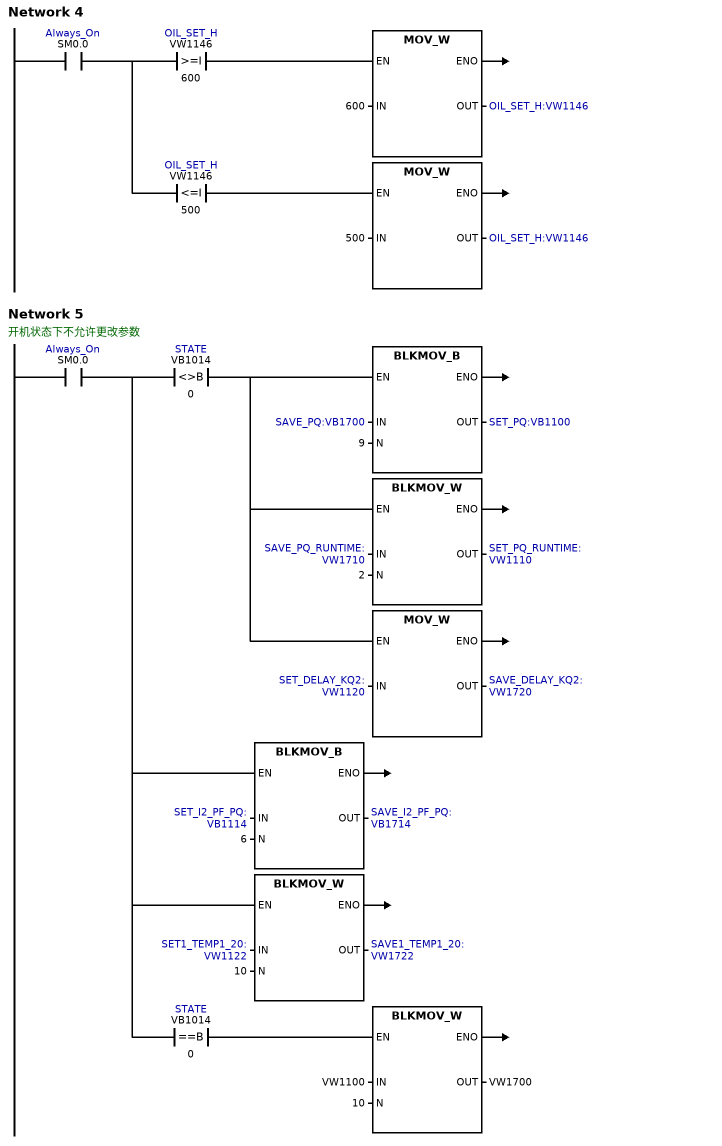
[picture p48: SBR5 networks 4-5]
Network 4
LD     Always_On:SM0.0
LPS
AW>=   OIL_SET_H:VW1146, 600
MOVW   600, OIL_SET_H:VW1146
LPP
AW<=   OIL_SET_H:VW1146, 500
MOVW   500, OIL_SET_H:VW1146
Network 5
// 开机状态下不允许更改参数
LD     Always_On:SM0.0
LPS
AB<>   STATE:VB1014, 0
BMB    SAVE_PQ:VB1700, SET_PQ:VB1100, 9
BMW    SAVE_PQ_RUNTIME:VW1710, SET_PQ_RUNTIME:VW1110, 2
MOVW   SET_DELAY_KQ2:VW1120, SAVE_DELAY_KQ2:VW1720
LPP
BMB    SET_I2_PF_PQ:VB1114, SAVE_I2_PF_PQ:VB1714, 6
BMW    SET1_TEMP1_20:VW1122, SAVE1_TEMP1_20:VW1722, 10
AB=    STATE:VB1014, 0
BMW    VW1100, VW1700, 10
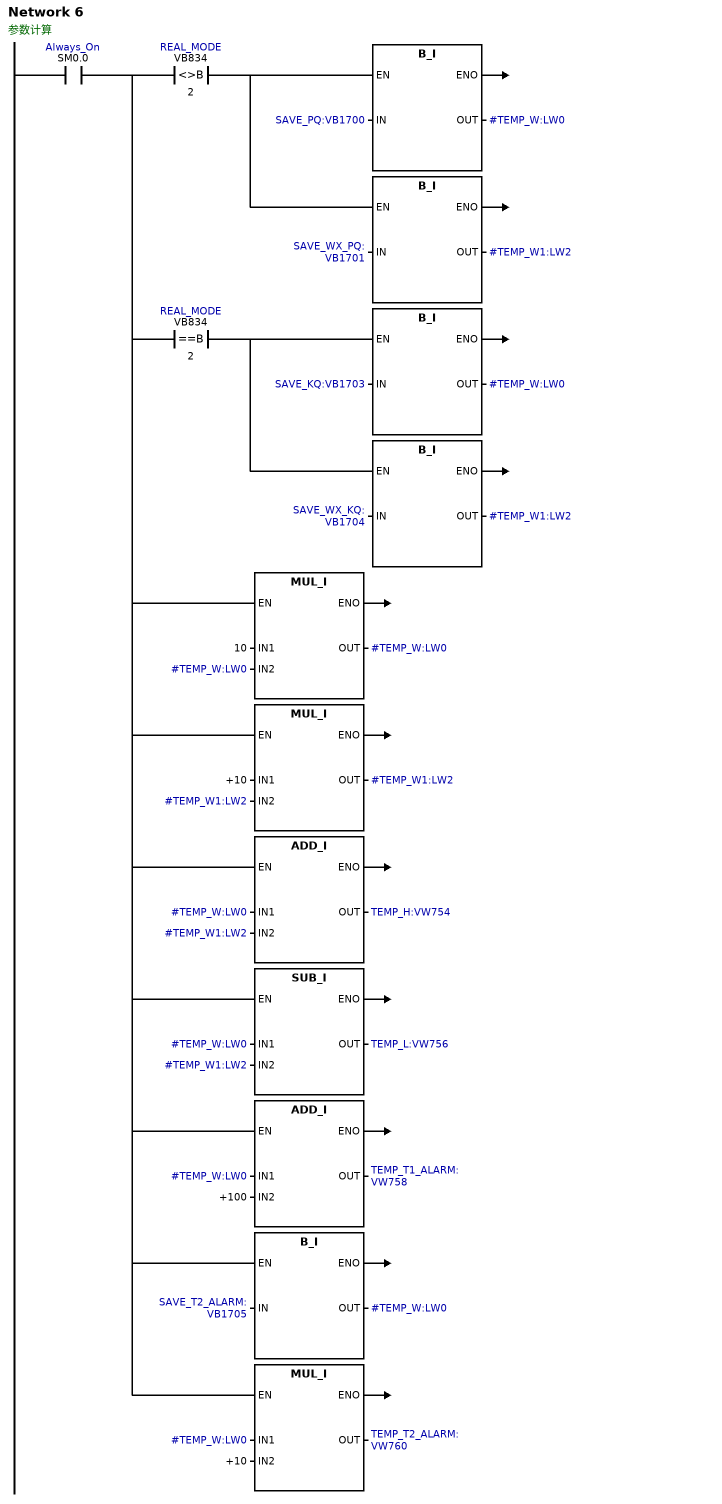
Network 6
// 参数计算
LD     Always_On:SM0.0
LPS
AB<>   REAL_MODE:VB834, 2
BTI    SAVE_PQ:VB1700, #TEMP_W:LW0
BTI    SAVE_WX_PQ:VB1701, #TEMP_W1:LW2
LRD
AB=    REAL_MODE:VB834, 2
BTI    SAVE_KQ:VB1703, #TEMP_W:LW0
BTI    SAVE_WX_KQ:VB1704, #TEMP_W1:LW2
LPP
*I     10, #TEMP_W:LW0
*I     +10, #TEMP_W1:LW2
MOVW   #TEMP_W:LW0, TEMP_H:VW754
+I     #TEMP_W1:LW2, TEMP_H:VW754
MOVW   #TEMP_W:LW0, TEMP_L:VW756
-I     #TEMP_W1:LW2, TEMP_L:VW756
MOVW   #TEMP_W:LW0, TEMP_T1_ALARM:VW758
+I     +100, TEMP_T1_ALARM:VW758
BTI    SAVE_T2_ALARM:VB1705, #TEMP_W:LW0
MOVW   #TEMP_W:LW0, TEMP_T2_ALARM:VW760
*I     +10, TEMP_T2_ALARM:VW760
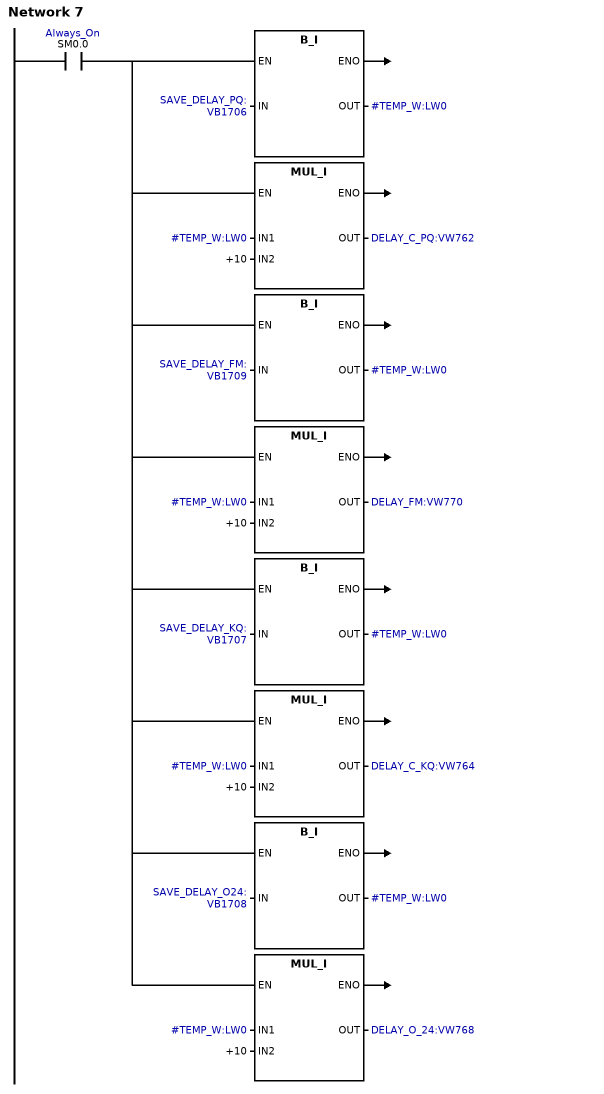
Network 7
LD     Always_On:SM0.0
BTI    SAVE_DELAY_PQ:VB1706, #TEMP_W:LW0
MOVW   #TEMP_W:LW0, DELAY_C_PQ:VW762
*I     +10, DELAY_C_PQ:VW762
BTI    SAVE_DELAY_FM:VB1709, #TEMP_W:LW0
MOVW   #TEMP_W:LW0, DELAY_FM:VW770
*I     +10, DELAY_FM:VW770
BTI    SAVE_DELAY_KQ:VB1707, #TEMP_W:LW0
MOVW   #TEMP_W:LW0, DELAY_C_KQ:VW764
*I     +10, DELAY_C_KQ:VW764
BTI    SAVE_DELAY_O24:VB1708, #TEMP_W:LW0
MOVW   #TEMP_W:LW0, DELAY_O_24:VW768
*I     +10, DELAY_O_24:VW768
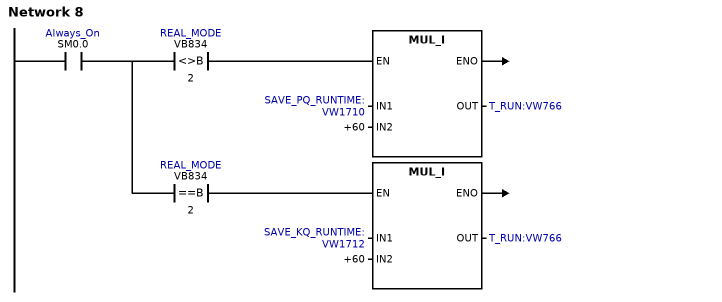
Network 8
LD     Always_On:SM0.0
LPS
AB<>   REAL_MODE:VB834, 2
MOVW   SAVE_PQ_RUNTIME:VW1710, T_RUN:VW766
*I     +60, T_RUN:VW766
LPP
AB=    REAL_MODE:VB834, 2
MOVW   SAVE_KQ_RUNTIME:VW1712, T_RUN:VW766
*I     +60, T_RUN:VW766
END_SUBROUTINE_BLOCK

SUBROUTINE_BLOCK 温度采样:SBR6
TITLE=
VAR_INPUT
ADDRESS:DWORD;	// LD0 
IN:WORD;	// LW4 
IN_TEMP:WORD;	// LW6 
F_SET:BOOL;	// L8.0 
END_VAR
VAR_OUTPUT
OUT:WORD;	// LW9 
AVERAGE:WORD;	// LW11 
OUT_TEMP:WORD;	// LW13 
END_VAR
VAR
MAX:WORD;	// LW15 
MIN:WORD;	// LW17 
TEMP_B:BYTE;	// LB19 
TEMP_W:WORD;	// LW20 
TEMP_DW:DWORD;	// LD22 
SUM:DWORD;	// LD26 
PP1:DWORD;	// LD30 
PP2:DWORD;	// LD34 
TEMP_W2:WORD;	// LW38 
AC_TEMP:DWORD;	// LD40 
END_VAR
BEGIN
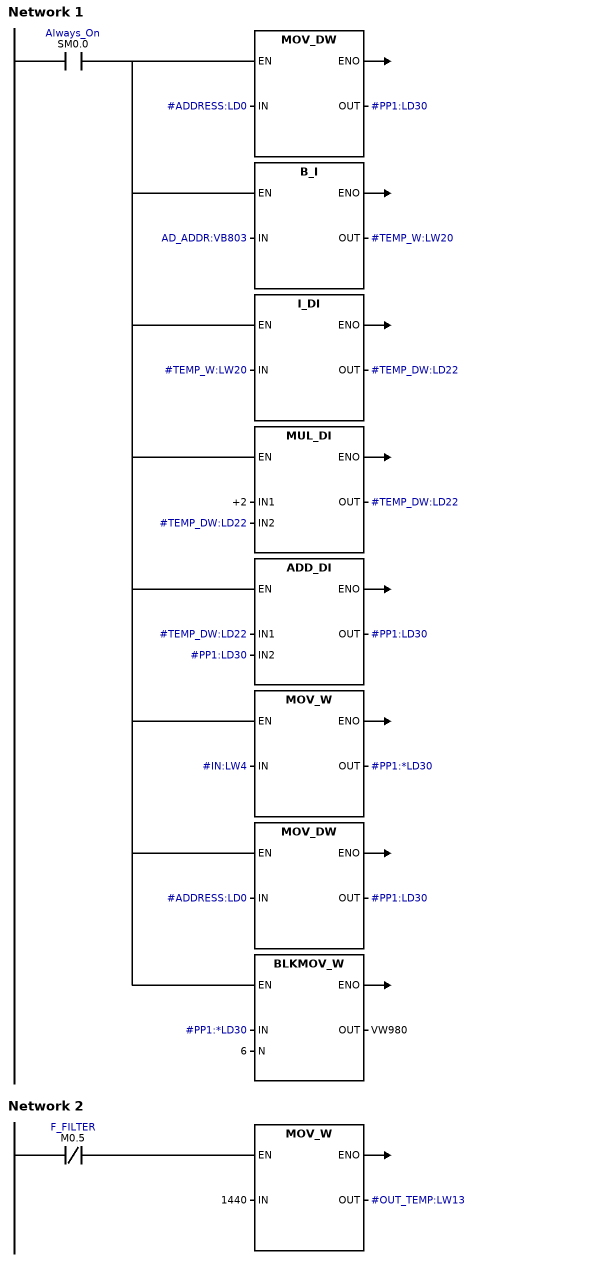
Network 1
LD     Always_On:SM0.0
MOVD   #ADDRESS:LD0, #PP1:LD30
BTI    AD_ADDR:VB803, #TEMP_W:LW20
ITD    #TEMP_W:LW20, #TEMP_DW:LD22
*D     +2, #TEMP_DW:LD22
+D     #TEMP_DW:LD22, #PP1:LD30
MOVW   #IN:LW4, *#PP1:LD30
MOVD   #ADDRESS:LD0, #PP1:LD30
BMW    *#PP1:LD30, VW980, 6
Network 2
LDN    F_FILTER:M0.5
MOVW   1440, #OUT_TEMP:LW13
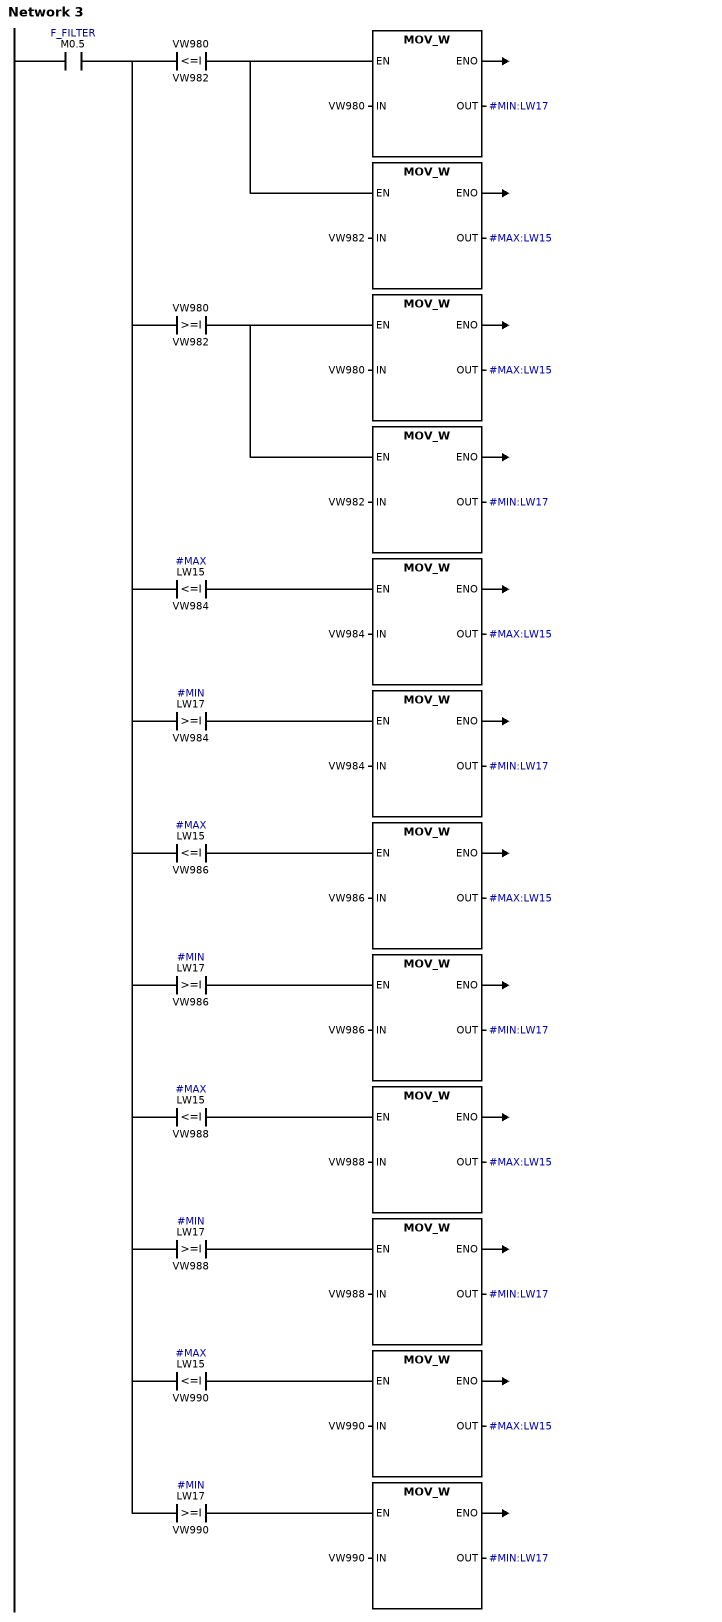
Network 3
LD     F_FILTER:M0.5
LPS
AW<=   VW980, VW982
MOVW   VW980, #MIN:LW17
MOVW   VW982, #MAX:LW15
LRD
AW>=   VW980, VW982
MOVW   VW980, #MAX:LW15
MOVW   VW982, #MIN:LW17
LPP
LPS
AW<=   #MAX:LW15, VW984
MOVW   VW984, #MAX:LW15
LRD
AW>=   #MIN:LW17, VW984
MOVW   VW984, #MIN:LW17
LRD
AW<=   #MAX:LW15, VW986
MOVW   VW986, #MAX:LW15
LRD
AW>=   #MIN:LW17, VW986
MOVW   VW986, #MIN:LW17
LRD
AW<=   #MAX:LW15, VW988
MOVW   VW988, #MAX:LW15
LRD
AW>=   #MIN:LW17, VW988
MOVW   VW988, #MIN:LW17
LRD
AW<=   #MAX:LW15, VW990
MOVW   VW990, #MAX:LW15
LPP
AW>=   #MIN:LW17, VW990
MOVW   VW990, #MIN:LW17
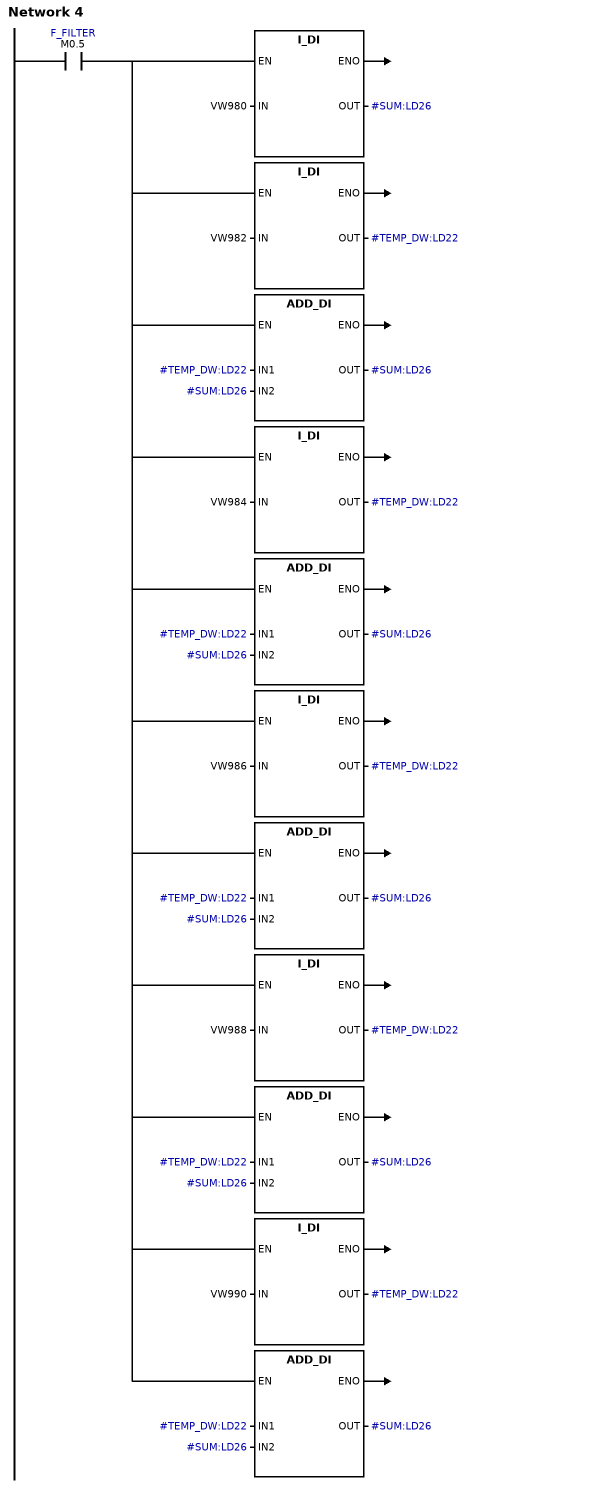
Network 4
LD     F_FILTER:M0.5
ITD    VW980, #SUM:LD26
ITD    VW982, #TEMP_DW:LD22
+D     #TEMP_DW:LD22, #SUM:LD26
ITD    VW984, #TEMP_DW:LD22
+D     #TEMP_DW:LD22, #SUM:LD26
ITD    VW986, #TEMP_DW:LD22
+D     #TEMP_DW:LD22, #SUM:LD26
ITD    VW988, #TEMP_DW:LD22
+D     #TEMP_DW:LD22, #SUM:LD26
ITD    VW990, #TEMP_DW:LD22
+D     #TEMP_DW:LD22, #SUM:LD26
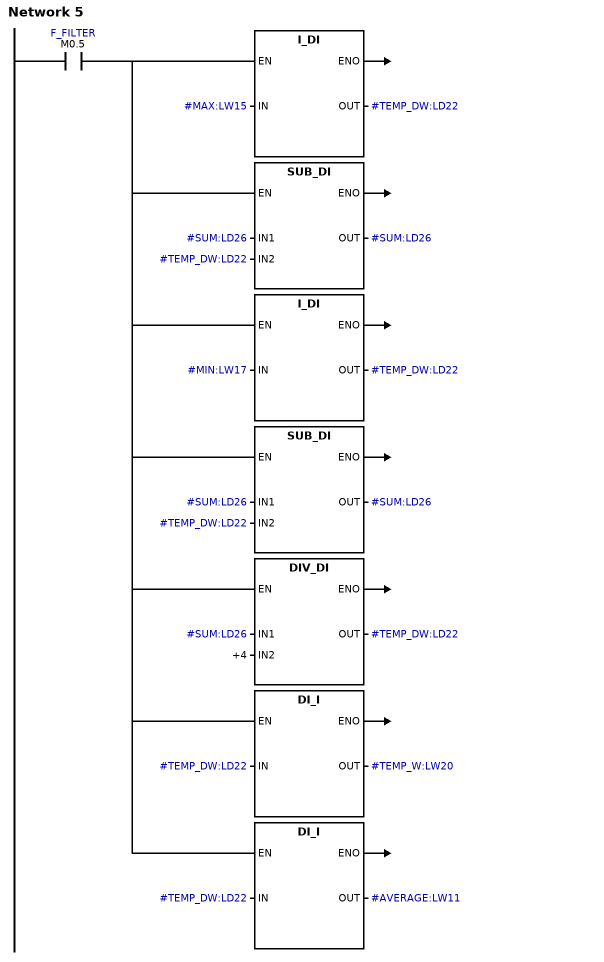
Network 5
LD     F_FILTER:M0.5
ITD    #MAX:LW15, #TEMP_DW:LD22
-D     #TEMP_DW:LD22, #SUM:LD26
ITD    #MIN:LW17, #TEMP_DW:LD22
-D     #TEMP_DW:LD22, #SUM:LD26
MOVD   #SUM:LD26, #TEMP_DW:LD22
/D     +4, #TEMP_DW:LD22
DTI    #TEMP_DW:LD22, #TEMP_W:LW20
DTI    #TEMP_DW:LD22, #AVERAGE:LW11
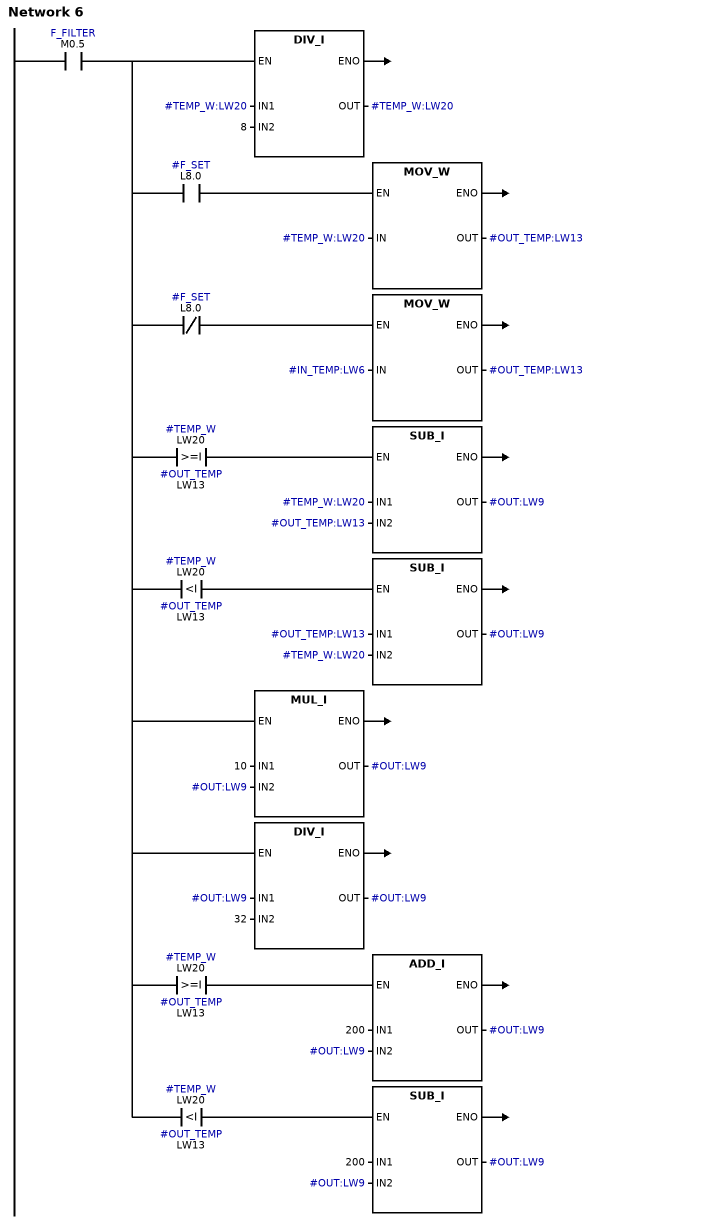
Network 6
LD     F_FILTER:M0.5
LPS
/I     8, #TEMP_W:LW20
A      #F_SET:L8.0
MOVW   #TEMP_W:LW20, #OUT_TEMP:LW13
LRD
AN     #F_SET:L8.0
MOVW   #IN_TEMP:LW6, #OUT_TEMP:LW13
LRD
AW>=   #TEMP_W:LW20, #OUT_TEMP:LW13
MOVW   #TEMP_W:LW20, #OUT:LW9
-I     #OUT_TEMP:LW13, #OUT:LW9
LRD
AW<    #TEMP_W:LW20, #OUT_TEMP:LW13
MOVW   #OUT_TEMP:LW13, #OUT:LW9
-I     #TEMP_W:LW20, #OUT:LW9
LRD
*I     10, #OUT:LW9
LRD
/I     32, #OUT:LW9
LRD
AW>=   #TEMP_W:LW20, #OUT_TEMP:LW13
+I     200, #OUT:LW9
LPP
AW<    #TEMP_W:LW20, #OUT_TEMP:LW13
INVW   #OUT:LW9
INCW   #OUT:LW9
+I     200, #OUT:LW9
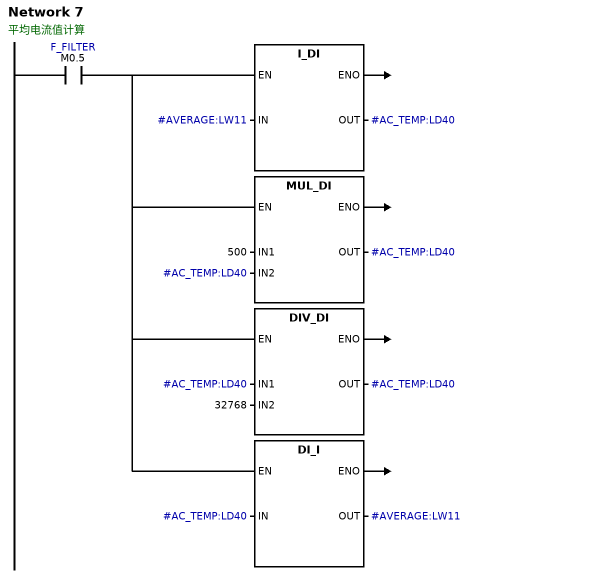
Network 7
// 平均电流值计算
LD     F_FILTER:M0.5
ITD    #AVERAGE:LW11, #AC_TEMP:LD40
*D     500, #AC_TEMP:LD40
/D     32768, #AC_TEMP:LD40
DTI    #AC_TEMP:LD40, #AVERAGE:LW11
END_SUBROUTINE_BLOCK

SUBROUTINE_BLOCK 启动停止控制:SBR7
TITLE=
BEGIN
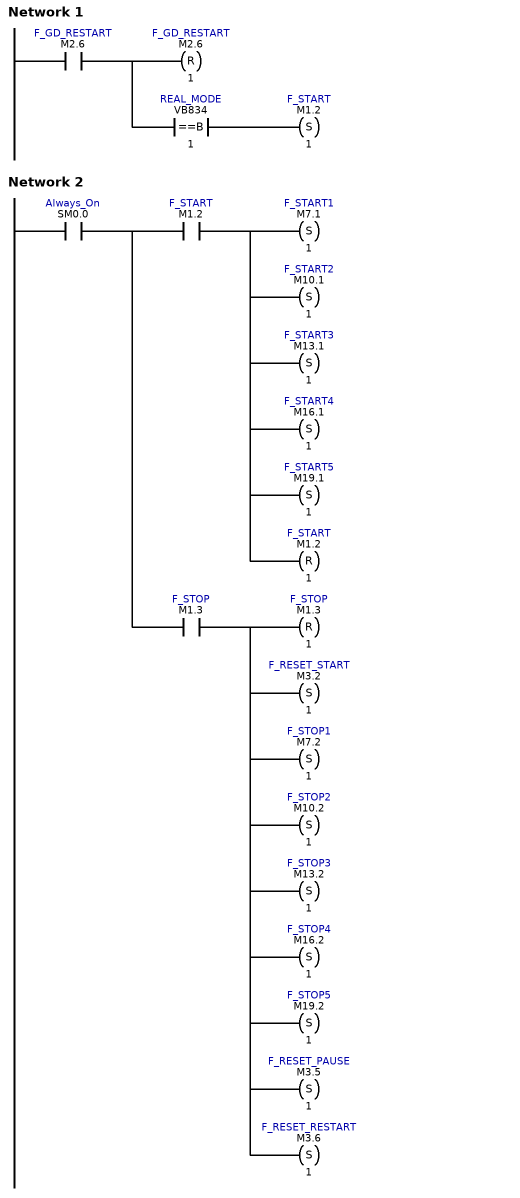
Network 1
LD     F_GD_RESTART:M2.6
R      F_GD_RESTART:M2.6, 1
AB=    REAL_MODE:VB834, 1
S      F_START:M1.2, 1
Network 2
LD     Always_On:SM0.0
LPS
A      F_START:M1.2
S      F_START1:M7.1, 1
S      F_START2:M10.1, 1
S      F_START3:M13.1, 1
S      F_START4:M16.1, 1
S      F_START5:M19.1, 1
R      F_START:M1.2, 1
LPP
A      F_STOP:M1.3
R      F_STOP:M1.3, 1
S      F_RESET_START:M3.2, 1
S      F_STOP1:M7.2, 1
S      F_STOP2:M10.2, 1
S      F_STOP3:M13.2, 1
S      F_STOP4:M16.2, 1
S      F_STOP5:M19.2, 1
S      F_RESET_PAUSE:M3.5, 1
S      F_RESET_RESTART:M3.6, 1
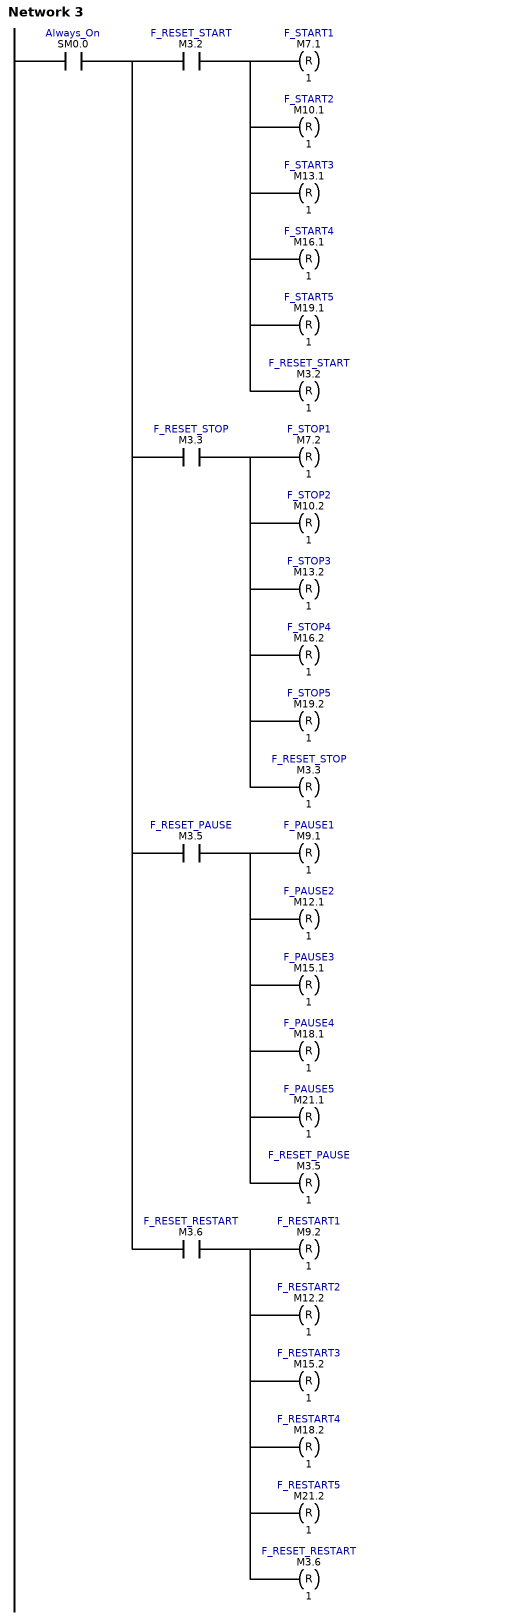
Network 3
LD     Always_On:SM0.0
LPS
A      F_RESET_START:M3.2
R      F_START1:M7.1, 1
R      F_START2:M10.1, 1
R      F_START3:M13.1, 1
R      F_START4:M16.1, 1
R      F_START5:M19.1, 1
R      F_RESET_START:M3.2, 1
LRD
A      F_RESET_STOP:M3.3
R      F_STOP1:M7.2, 1
R      F_STOP2:M10.2, 1
R      F_STOP3:M13.2, 1
R      F_STOP4:M16.2, 1
R      F_STOP5:M19.2, 1
R      F_RESET_STOP:M3.3, 1
LRD
A      F_RESET_PAUSE:M3.5
R      F_PAUSE1:M9.1, 1
R      F_PAUSE2:M12.1, 1
R      F_PAUSE3:M15.1, 1
R      F_PAUSE4:M18.1, 1
R      F_PAUSE5:M21.1, 1
R      F_RESET_PAUSE:M3.5, 1
LPP
A      F_RESET_RESTART:M3.6
R      F_RESTART1:M9.2, 1
R      F_RESTART2:M12.2, 1
R      F_RESTART3:M15.2, 1
R      F_RESTART4:M18.2, 1
R      F_RESTART5:M21.2, 1
R      F_RESET_RESTART:M3.6, 1
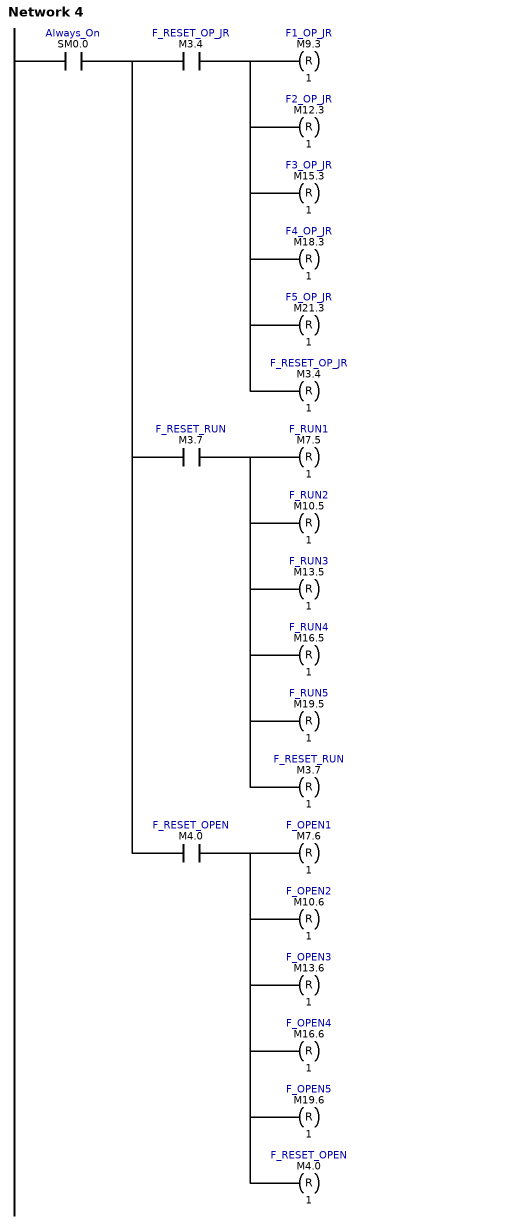
Network 4
LD     Always_On:SM0.0
LPS
A      F_RESET_OP_JR:M3.4
R      F1_OP_JR:M9.3, 1
R      F2_OP_JR:M12.3, 1
R      F3_OP_JR:M15.3, 1
R      F4_OP_JR:M18.3, 1
R      F5_OP_JR:M21.3, 1
R      F_RESET_OP_JR:M3.4, 1
LRD
A      F_RESET_RUN:M3.7
R      F_RUN1:M7.5, 1
R      F_RUN2:M10.5, 1
R      F_RUN3:M13.5, 1
R      F_RUN4:M16.5, 1
R      F_RUN5:M19.5, 1
R      F_RESET_RUN:M3.7, 1
LPP
A      F_RESET_OPEN:M4.0
R      F_OPEN1:M7.6, 1
R      F_OPEN2:M10.6, 1
R      F_OPEN3:M13.6, 1
R      F_OPEN4:M16.6, 1
R      F_OPEN5:M19.6, 1
R      F_RESET_OPEN:M4.0, 1
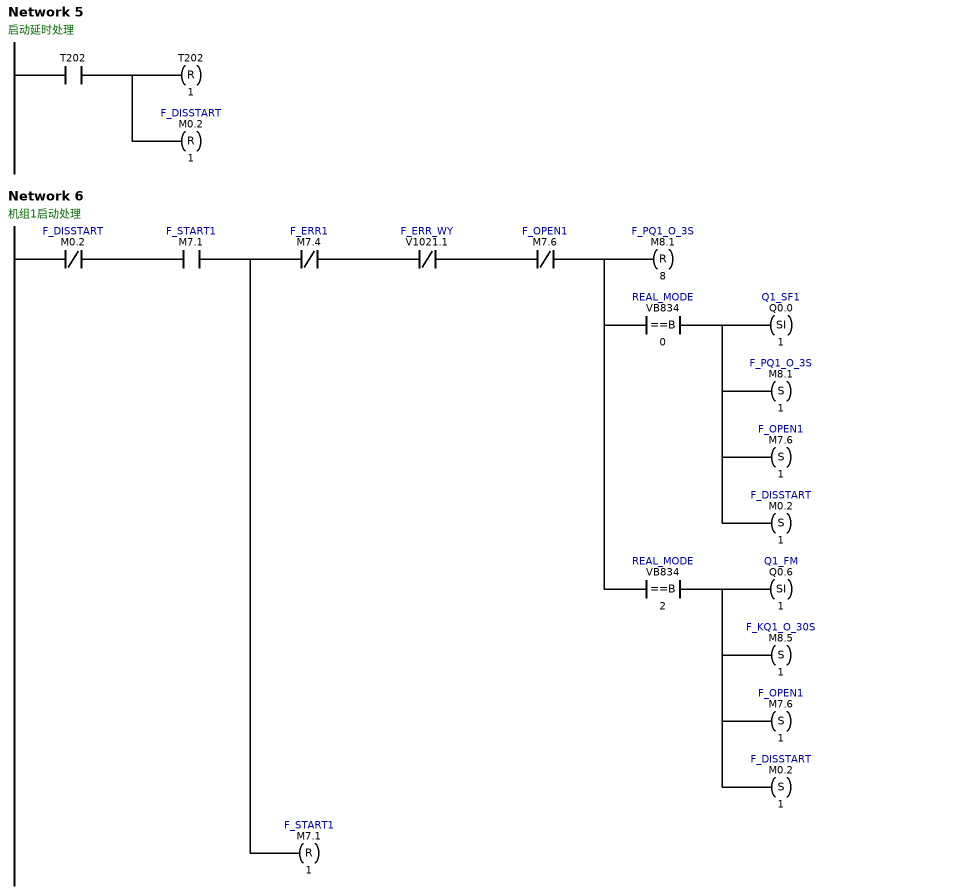
Network 5
// 启动延时处理
LD     T202
R      T202, 1
R      F_DISSTART:M0.2, 1
Network 6
// 机组1启动处理
LDN    F_DISSTART:M0.2
A      F_START1:M7.1
LPS
AN     F_ERR1:M7.4
AN     F_ERR_WY:V1021.1
AN     F_OPEN1:M7.6
LPS
R      F_PQ1_O_3S:M8.1, 8
AB=    REAL_MODE:VB834, 0
SI     Q1_SF1:Q0.0, 1
S      F_PQ1_O_3S:M8.1, 1
S      F_OPEN1:M7.6, 1
S      F_DISSTART:M0.2, 1
LPP
AB=    REAL_MODE:VB834, 2
SI     Q1_FM:Q0.6, 1
S      F_KQ1_O_30S:M8.5, 1
S      F_OPEN1:M7.6, 1
S      F_DISSTART:M0.2, 1
LPP
R      F_START1:M7.1, 1
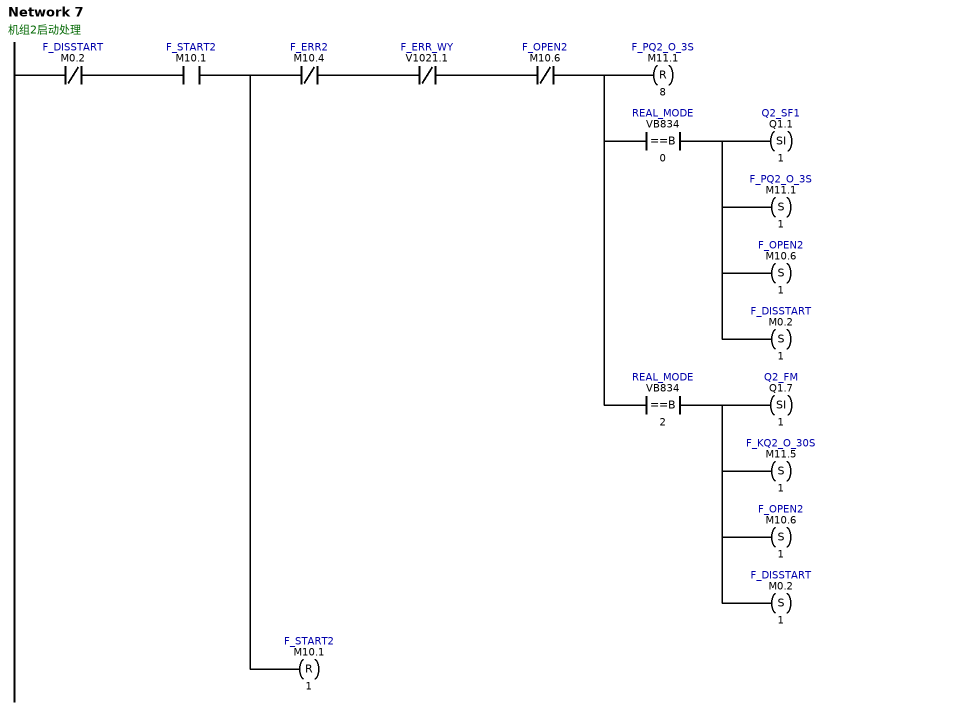
Network 7
// 机组2启动处理
LDN    F_DISSTART:M0.2
A      F_START2:M10.1
LPS
AN     F_ERR2:M10.4
AN     F_ERR_WY:V1021.1
AN     F_OPEN2:M10.6
LPS
R      F_PQ2_O_3S:M11.1, 8
AB=    REAL_MODE:VB834, 0
SI     Q2_SF1:Q1.1, 1
S      F_PQ2_O_3S:M11.1, 1
S      F_OPEN2:M10.6, 1
S      F_DISSTART:M0.2, 1
LPP
AB=    REAL_MODE:VB834, 2
SI     Q2_FM:Q1.7, 1
S      F_KQ2_O_30S:M11.5, 1
S      F_OPEN2:M10.6, 1
S      F_DISSTART:M0.2, 1
LPP
R      F_START2:M10.1, 1
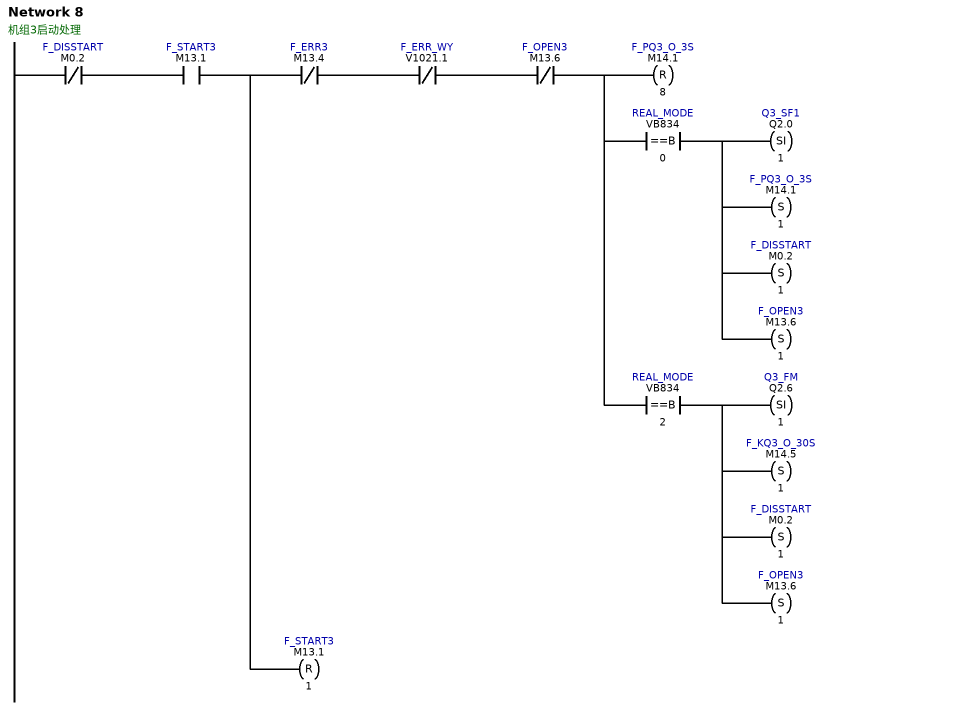
Network 8
// 机组3启动处理
LDN    F_DISSTART:M0.2
A      F_START3:M13.1
LPS
AN     F_ERR3:M13.4
AN     F_ERR_WY:V1021.1
AN     F_OPEN3:M13.6
LPS
R      F_PQ3_O_3S:M14.1, 8
AB=    REAL_MODE:VB834, 0
SI     Q3_SF1:Q2.0, 1
S      F_PQ3_O_3S:M14.1, 1
S      F_DISSTART:M0.2, 1
S      F_OPEN3:M13.6, 1
LPP
AB=    REAL_MODE:VB834, 2
SI     Q3_FM:Q2.6, 1
S      F_KQ3_O_30S:M14.5, 1
S      F_DISSTART:M0.2, 1
S      F_OPEN3:M13.6, 1
LPP
R      F_START3:M13.1, 1
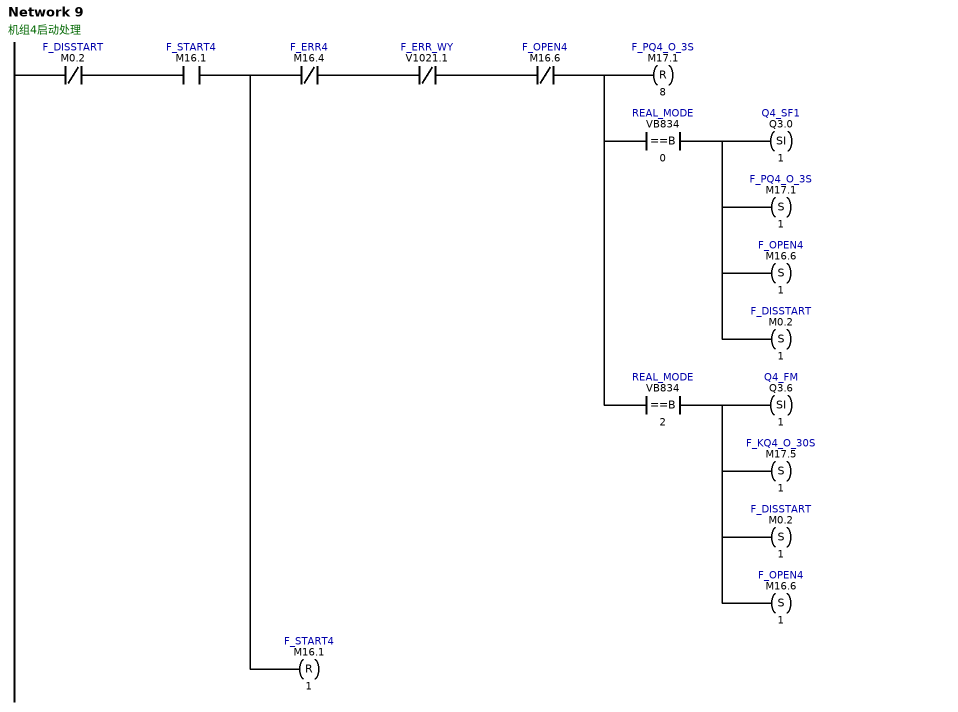
Network 9
// 机组4启动处理
LDN    F_DISSTART:M0.2
A      F_START4:M16.1
LPS
AN     F_ERR4:M16.4
AN     F_ERR_WY:V1021.1
AN     F_OPEN4:M16.6
LPS
R      F_PQ4_O_3S:M17.1, 8
AB=    REAL_MODE:VB834, 0
SI     Q4_SF1:Q3.0, 1
S      F_PQ4_O_3S:M17.1, 1
S      F_OPEN4:M16.6, 1
S      F_DISSTART:M0.2, 1
LPP
AB=    REAL_MODE:VB834, 2
SI     Q4_FM:Q3.6, 1
S      F_KQ4_O_30S:M17.5, 1
S      F_DISSTART:M0.2, 1
S      F_OPEN4:M16.6, 1
LPP
R      F_START4:M16.1, 1
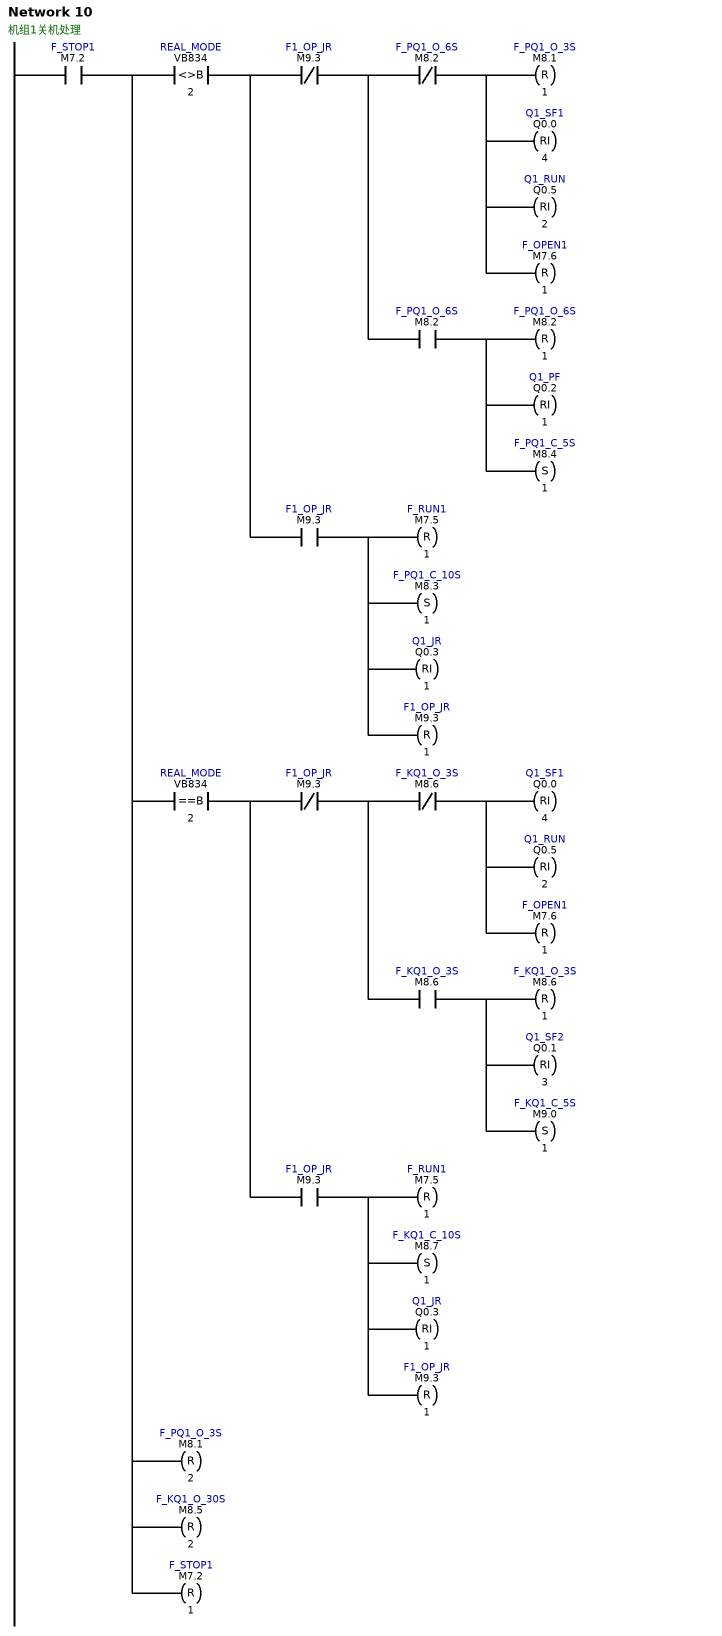
Network 10
// 机组1关机处理
LD     F_STOP1:M7.2
LPS
AB<>   REAL_MODE:VB834, 2
LPS
AN     F1_OP_JR:M9.3
LPS
AN     F_PQ1_O_6S:M8.2
R      F_PQ1_O_3S:M8.1, 1
RI     Q1_SF1:Q0.0, 4
RI     Q1_RUN:Q0.5, 2
R      F_OPEN1:M7.6, 1
LPP
A      F_PQ1_O_6S:M8.2
R      F_PQ1_O_6S:M8.2, 1
RI     Q1_PF:Q0.2, 1
S      F_PQ1_C_5S:M8.4, 1
LPP
A      F1_OP_JR:M9.3
R      F_RUN1:M7.5, 1
S      F_PQ1_C_10S:M8.3, 1
RI     Q1_JR:Q0.3, 1
R      F1_OP_JR:M9.3, 1
LRD
AB=    REAL_MODE:VB834, 2
LPS
AN     F1_OP_JR:M9.3
LPS
AN     F_KQ1_O_3S:M8.6
RI     Q1_SF1:Q0.0, 4
RI     Q1_RUN:Q0.5, 2
R      F_OPEN1:M7.6, 1
LPP
A      F_KQ1_O_3S:M8.6
R      F_KQ1_O_3S:M8.6, 1
RI     Q1_SF2:Q0.1, 3
S      F_KQ1_C_5S:M9.0, 1
LPP
A      F1_OP_JR:M9.3
R      F_RUN1:M7.5, 1
S      F_KQ1_C_10S:M8.7, 1
RI     Q1_JR:Q0.3, 1
R      F1_OP_JR:M9.3, 1
LPP
R      F_PQ1_O_3S:M8.1, 2
R      F_KQ1_O_30S:M8.5, 2
R      F_STOP1:M7.2, 1
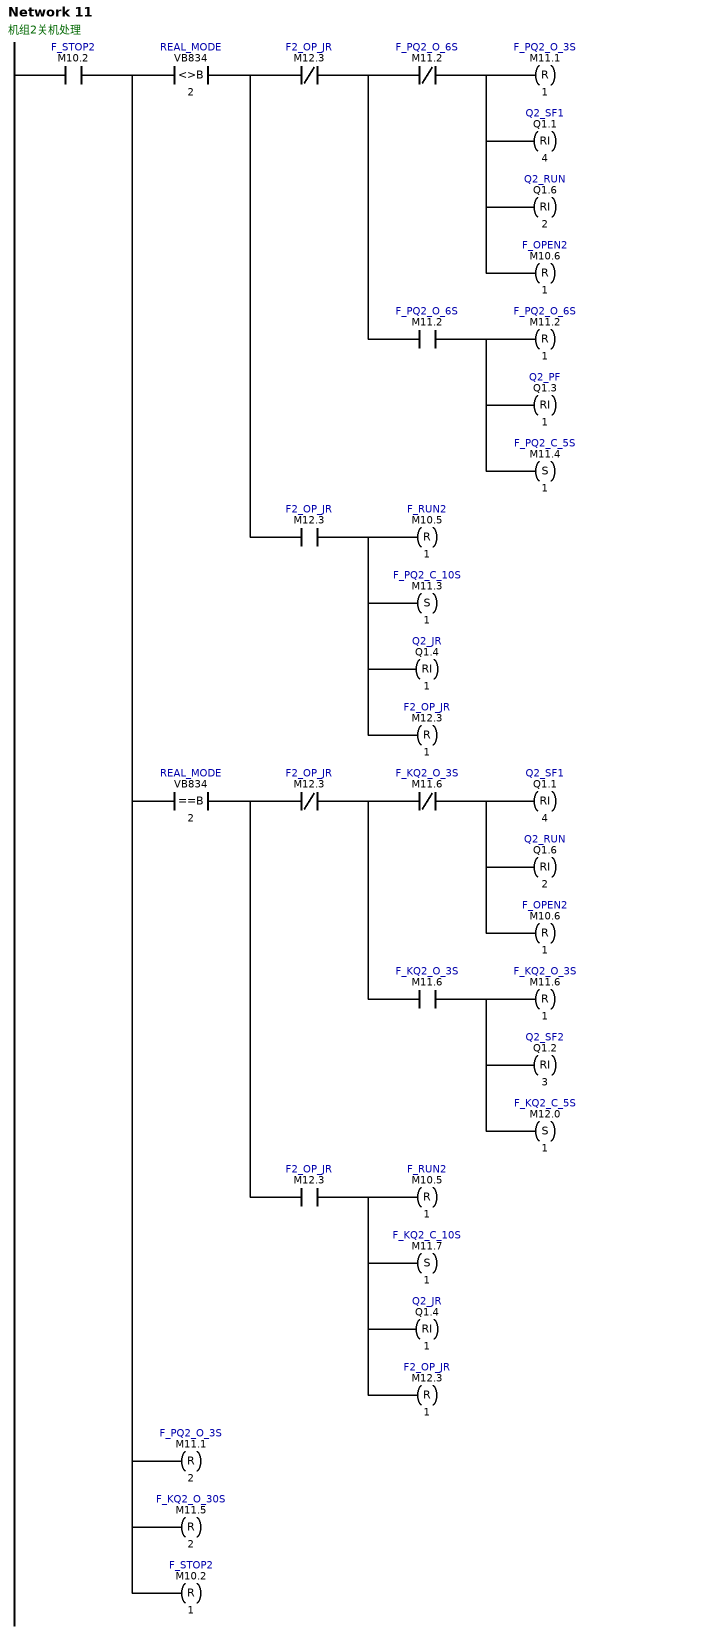
Network 11
// 机组2关机处理
LD     F_STOP2:M10.2
LPS
AB<>   REAL_MODE:VB834, 2
LPS
AN     F2_OP_JR:M12.3
LPS
AN     F_PQ2_O_6S:M11.2
R      F_PQ2_O_3S:M11.1, 1
RI     Q2_SF1:Q1.1, 4
RI     Q2_RUN:Q1.6, 2
R      F_OPEN2:M10.6, 1
LPP
A      F_PQ2_O_6S:M11.2
R      F_PQ2_O_6S:M11.2, 1
RI     Q2_PF:Q1.3, 1
S      F_PQ2_C_5S:M11.4, 1
LPP
A      F2_OP_JR:M12.3
R      F_RUN2:M10.5, 1
S      F_PQ2_C_10S:M11.3, 1
RI     Q2_JR:Q1.4, 1
R      F2_OP_JR:M12.3, 1
LRD
AB=    REAL_MODE:VB834, 2
LPS
AN     F2_OP_JR:M12.3
LPS
AN     F_KQ2_O_3S:M11.6
RI     Q2_SF1:Q1.1, 4
RI     Q2_RUN:Q1.6, 2
R      F_OPEN2:M10.6, 1
LPP
A      F_KQ2_O_3S:M11.6
R      F_KQ2_O_3S:M11.6, 1
RI     Q2_SF2:Q1.2, 3
S      F_KQ2_C_5S:M12.0, 1
LPP
A      F2_OP_JR:M12.3
R      F_RUN2:M10.5, 1
S      F_KQ2_C_10S:M11.7, 1
RI     Q2_JR:Q1.4, 1
R      F2_OP_JR:M12.3, 1
LPP
R      F_PQ2_O_3S:M11.1, 2
R      F_KQ2_O_30S:M11.5, 2
R      F_STOP2:M10.2, 1
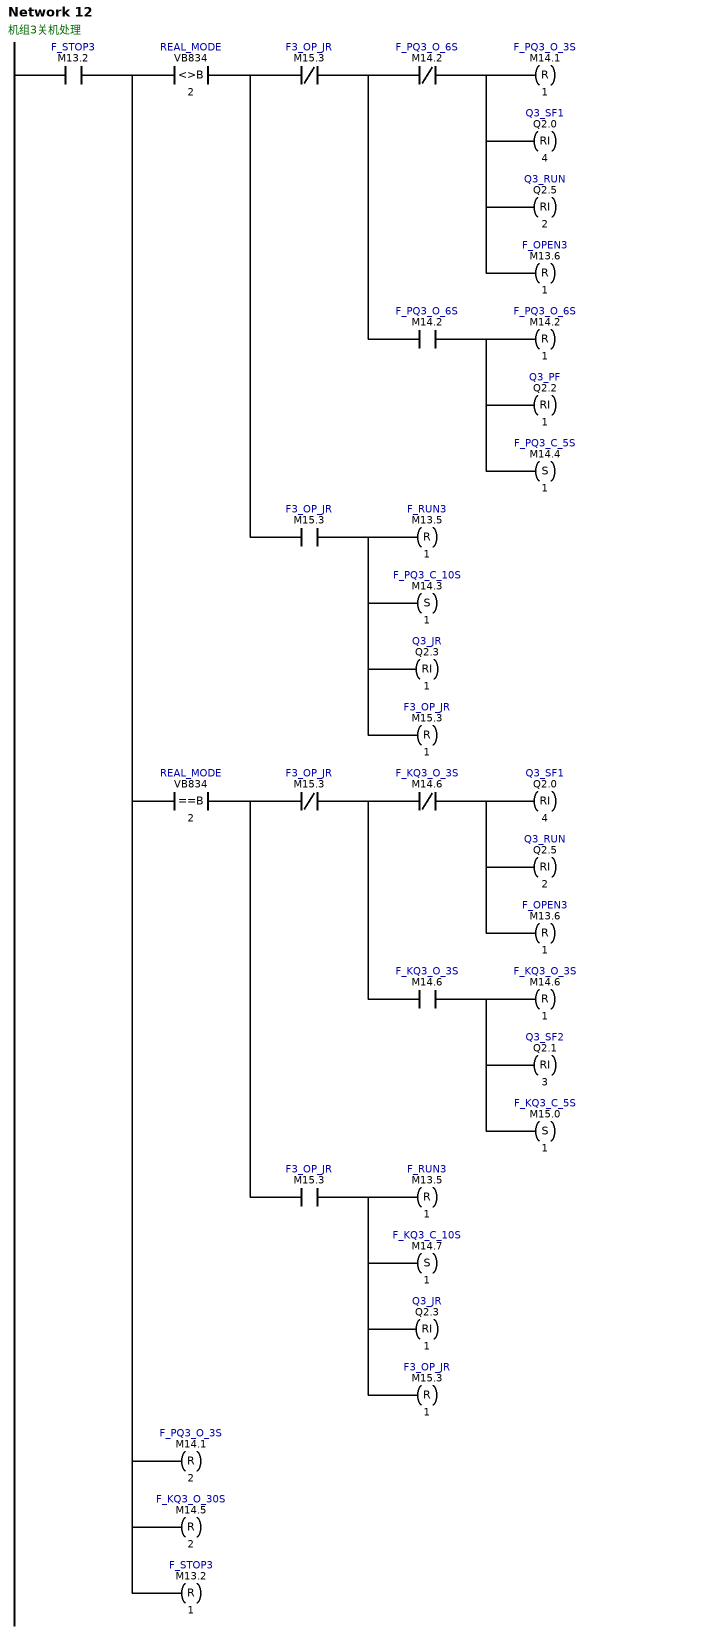
Network 12
// 机组3关机处理
LD     F_STOP3:M13.2
LPS
AB<>   REAL_MODE:VB834, 2
LPS
AN     F3_OP_JR:M15.3
LPS
AN     F_PQ3_O_6S:M14.2
R      F_PQ3_O_3S:M14.1, 1
RI     Q3_SF1:Q2.0, 4
RI     Q3_RUN:Q2.5, 2
R      F_OPEN3:M13.6, 1
LPP
A      F_PQ3_O_6S:M14.2
R      F_PQ3_O_6S:M14.2, 1
RI     Q3_PF:Q2.2, 1
S      F_PQ3_C_5S:M14.4, 1
LPP
A      F3_OP_JR:M15.3
R      F_RUN3:M13.5, 1
S      F_PQ3_C_10S:M14.3, 1
RI     Q3_JR:Q2.3, 1
R      F3_OP_JR:M15.3, 1
LRD
AB=    REAL_MODE:VB834, 2
LPS
AN     F3_OP_JR:M15.3
LPS
AN     F_KQ3_O_3S:M14.6
RI     Q3_SF1:Q2.0, 4
RI     Q3_RUN:Q2.5, 2
R      F_OPEN3:M13.6, 1
LPP
A      F_KQ3_O_3S:M14.6
R      F_KQ3_O_3S:M14.6, 1
RI     Q3_SF2:Q2.1, 3
S      F_KQ3_C_5S:M15.0, 1
LPP
A      F3_OP_JR:M15.3
R      F_RUN3:M13.5, 1
S      F_KQ3_C_10S:M14.7, 1
RI     Q3_JR:Q2.3, 1
R      F3_OP_JR:M15.3, 1
LPP
R      F_PQ3_O_3S:M14.1, 2
R      F_KQ3_O_30S:M14.5, 2
R      F_STOP3:M13.2, 1
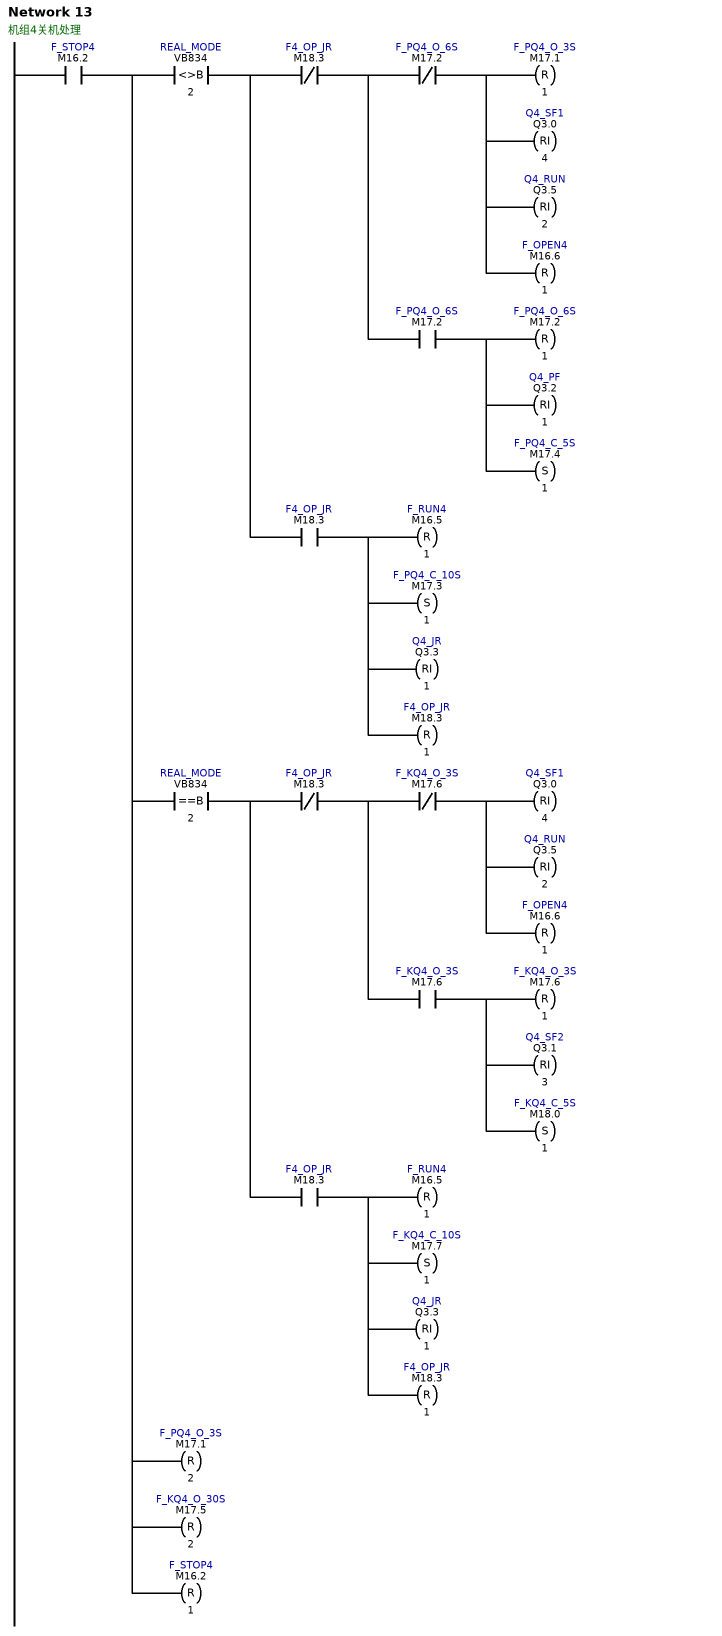
Network 13
// 机组4关机处理
LD     F_STOP4:M16.2
LPS
AB<>   REAL_MODE:VB834, 2
LPS
AN     F4_OP_JR:M18.3
LPS
AN     F_PQ4_O_6S:M17.2
R      F_PQ4_O_3S:M17.1, 1
RI     Q4_SF1:Q3.0, 4
RI     Q4_RUN:Q3.5, 2
R      F_OPEN4:M16.6, 1
LPP
A      F_PQ4_O_6S:M17.2
R      F_PQ4_O_6S:M17.2, 1
RI     Q4_PF:Q3.2, 1
S      F_PQ4_C_5S:M17.4, 1
LPP
A      F4_OP_JR:M18.3
R      F_RUN4:M16.5, 1
S      F_PQ4_C_10S:M17.3, 1
RI     Q4_JR:Q3.3, 1
R      F4_OP_JR:M18.3, 1
LRD
AB=    REAL_MODE:VB834, 2
LPS
AN     F4_OP_JR:M18.3
LPS
AN     F_KQ4_O_3S:M17.6
RI     Q4_SF1:Q3.0, 4
RI     Q4_RUN:Q3.5, 2
R      F_OPEN4:M16.6, 1
LPP
A      F_KQ4_O_3S:M17.6
R      F_KQ4_O_3S:M17.6, 1
RI     Q4_SF2:Q3.1, 3
S      F_KQ4_C_5S:M18.0, 1
LPP
A      F4_OP_JR:M18.3
R      F_RUN4:M16.5, 1
S      F_KQ4_C_10S:M17.7, 1
RI     Q4_JR:Q3.3, 1
R      F4_OP_JR:M18.3, 1
LPP
R      F_PQ4_O_3S:M17.1, 2
R      F_KQ4_O_30S:M17.5, 2
R      F_STOP4:M16.2, 1
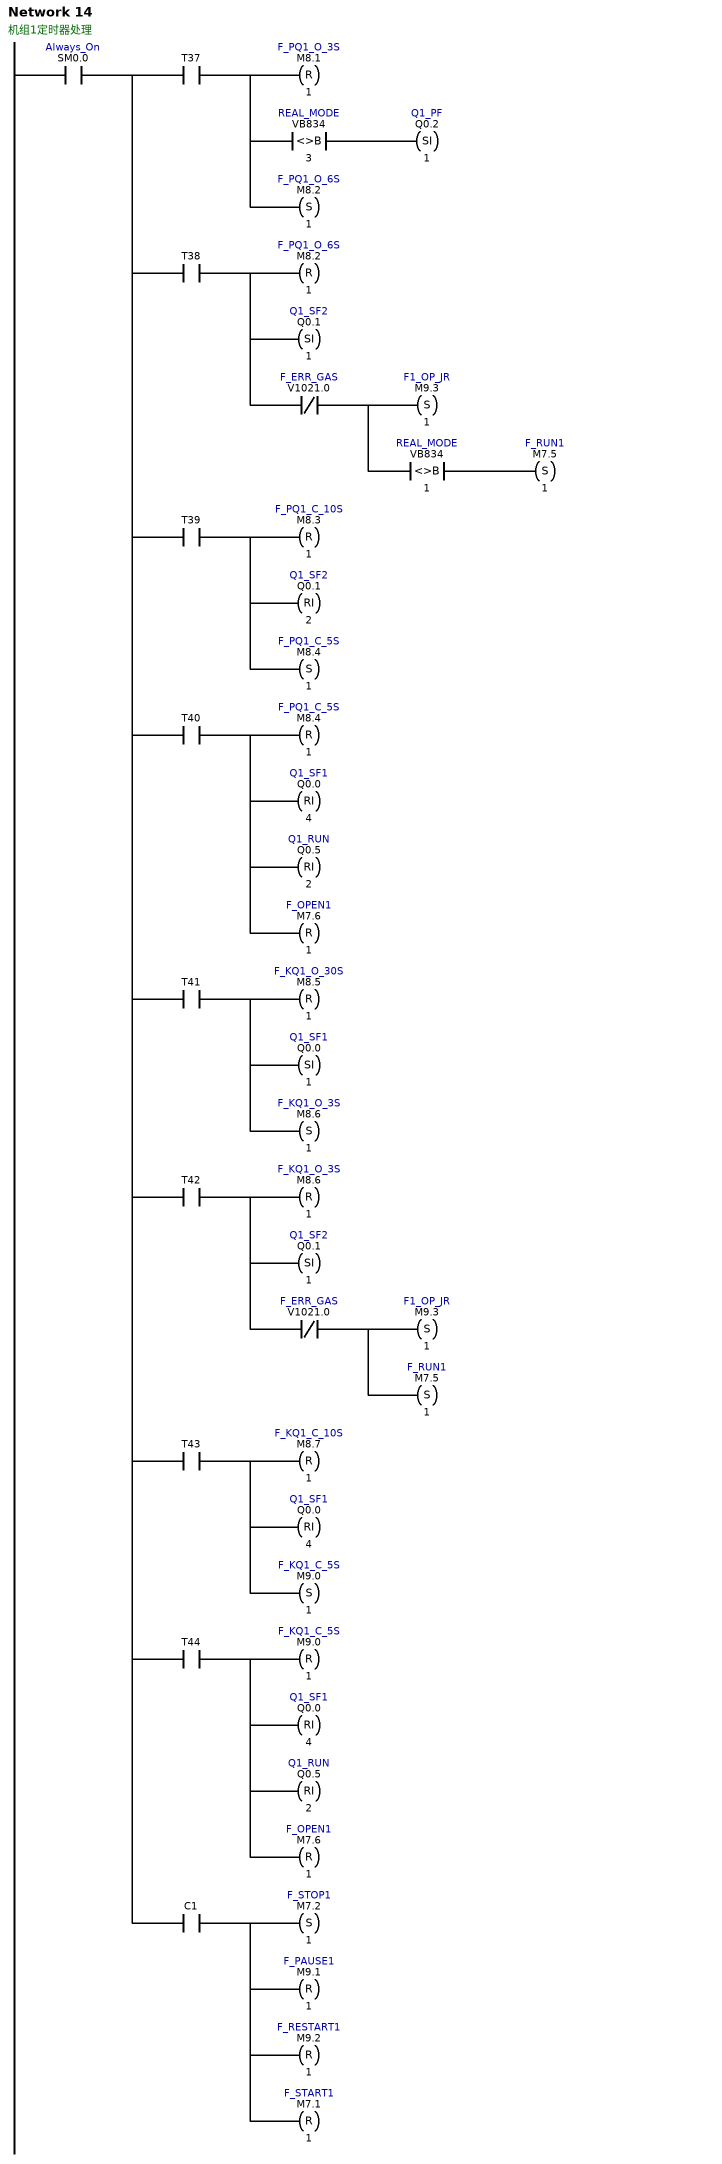
Network 14
// 机组1定时器处理
LD     Always_On:SM0.0
LPS
A      T37
LPS
R      F_PQ1_O_3S:M8.1, 1
AB<>   REAL_MODE:VB834, 3
SI     Q1_PF:Q0.2, 1
LPP
S      F_PQ1_O_6S:M8.2, 1
LRD
A      T38
R      F_PQ1_O_6S:M8.2, 1
SI     Q1_SF2:Q0.1, 1
AN     F_ERR_GAS:V1021.0
S      F1_OP_JR:M9.3, 1
AB<>   REAL_MODE:VB834, 1
S      F_RUN1:M7.5, 1
LRD
LPS
A      T39
R      F_PQ1_C_10S:M8.3, 1
RI     Q1_SF2:Q0.1, 2
S      F_PQ1_C_5S:M8.4, 1
LRD
A      T40
R      F_PQ1_C_5S:M8.4, 1
RI     Q1_SF1:Q0.0, 4
RI     Q1_RUN:Q0.5, 2
R      F_OPEN1:M7.6, 1
LPP
A      T41
R      F_KQ1_O_30S:M8.5, 1
SI     Q1_SF1:Q0.0, 1
S      F_KQ1_O_3S:M8.6, 1
LRD
A      T42
R      F_KQ1_O_3S:M8.6, 1
SI     Q1_SF2:Q0.1, 1
AN     F_ERR_GAS:V1021.0
S      F1_OP_JR:M9.3, 1
S      F_RUN1:M7.5, 1
LPP
LPS
A      T43
R      F_KQ1_C_10S:M8.7, 1
RI     Q1_SF1:Q0.0, 4
S      F_KQ1_C_5S:M9.0, 1
LRD
A      T44
R      F_KQ1_C_5S:M9.0, 1
RI     Q1_SF1:Q0.0, 4
RI     Q1_RUN:Q0.5, 2
R      F_OPEN1:M7.6, 1
LPP
A      C1
S      F_STOP1:M7.2, 1
R      F_PAUSE1:M9.1, 1
R      F_RESTART1:M9.2, 1
R      F_START1:M7.1, 1
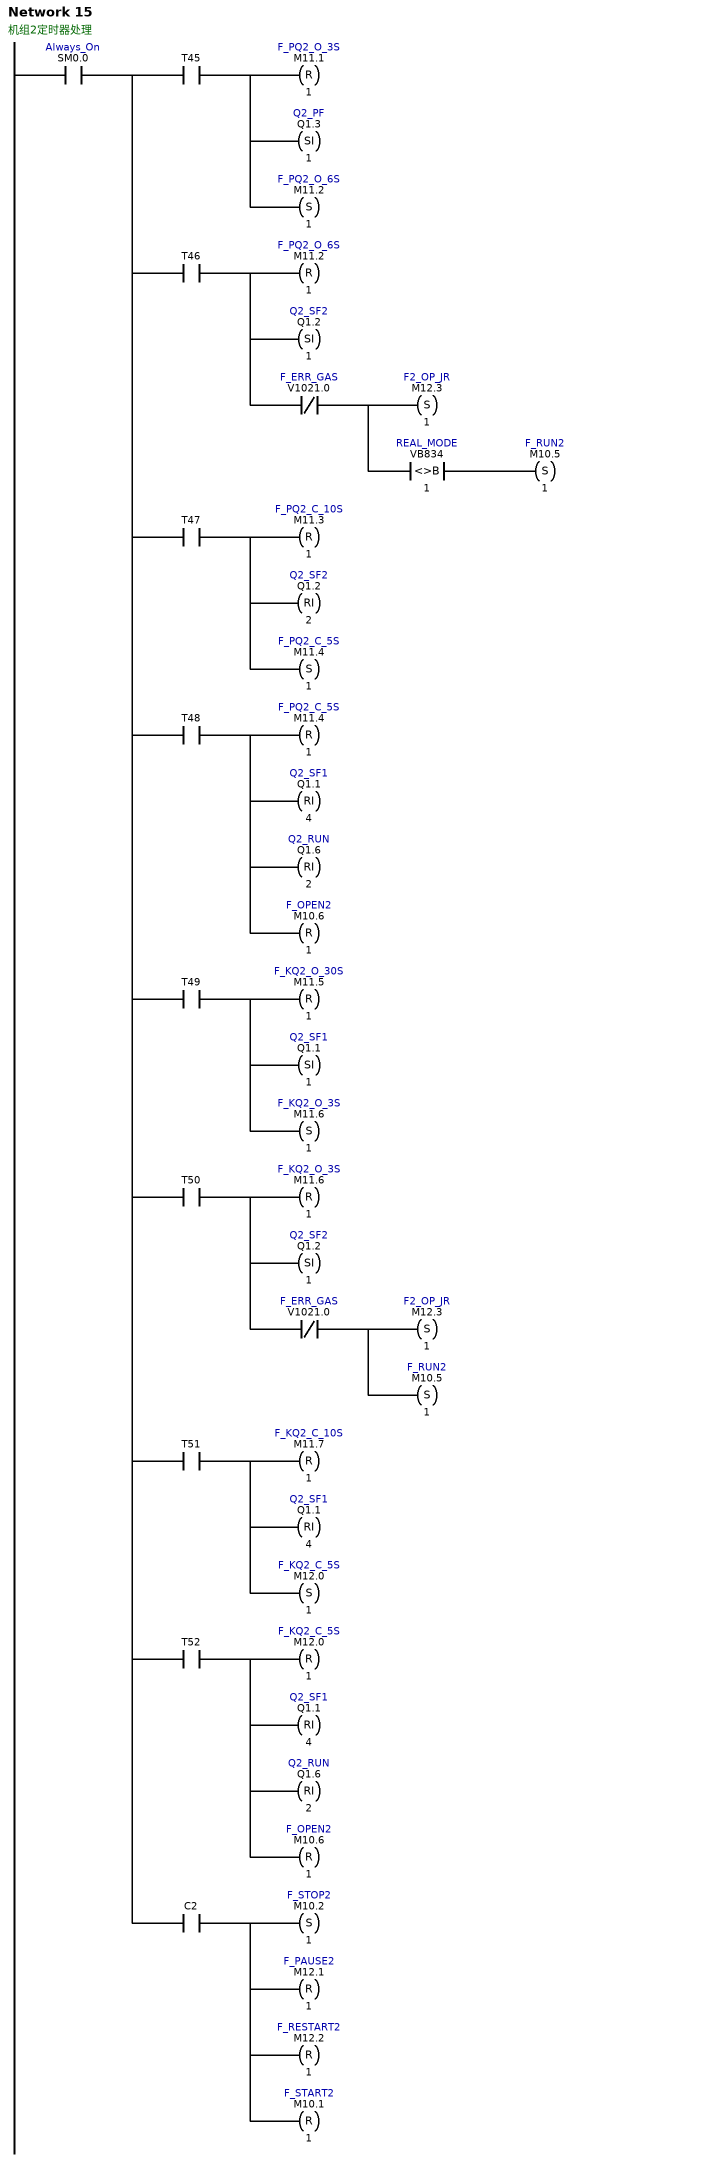
Network 15
// 机组2定时器处理
LD     Always_On:SM0.0
LPS
A      T45
R      F_PQ2_O_3S:M11.1, 1
SI     Q2_PF:Q1.3, 1
S      F_PQ2_O_6S:M11.2, 1
LRD
A      T46
R      F_PQ2_O_6S:M11.2, 1
SI     Q2_SF2:Q1.2, 1
AN     F_ERR_GAS:V1021.0
S      F2_OP_JR:M12.3, 1
AB<>   REAL_MODE:VB834, 1
S      F_RUN2:M10.5, 1
LRD
LPS
A      T47
R      F_PQ2_C_10S:M11.3, 1
RI     Q2_SF2:Q1.2, 2
S      F_PQ2_C_5S:M11.4, 1
LRD
A      T48
R      F_PQ2_C_5S:M11.4, 1
RI     Q2_SF1:Q1.1, 4
RI     Q2_RUN:Q1.6, 2
R      F_OPEN2:M10.6, 1
LPP
A      T49
R      F_KQ2_O_30S:M11.5, 1
SI     Q2_SF1:Q1.1, 1
S      F_KQ2_O_3S:M11.6, 1
LRD
A      T50
R      F_KQ2_O_3S:M11.6, 1
SI     Q2_SF2:Q1.2, 1
AN     F_ERR_GAS:V1021.0
S      F2_OP_JR:M12.3, 1
S      F_RUN2:M10.5, 1
LPP
LPS
A      T51
R      F_KQ2_C_10S:M11.7, 1
RI     Q2_SF1:Q1.1, 4
S      F_KQ2_C_5S:M12.0, 1
LRD
A      T52
R      F_KQ2_C_5S:M12.0, 1
RI     Q2_SF1:Q1.1, 4
RI     Q2_RUN:Q1.6, 2
R      F_OPEN2:M10.6, 1
LPP
A      C2
S      F_STOP2:M10.2, 1
R      F_PAUSE2:M12.1, 1
R      F_RESTART2:M12.2, 1
R      F_START2:M10.1, 1
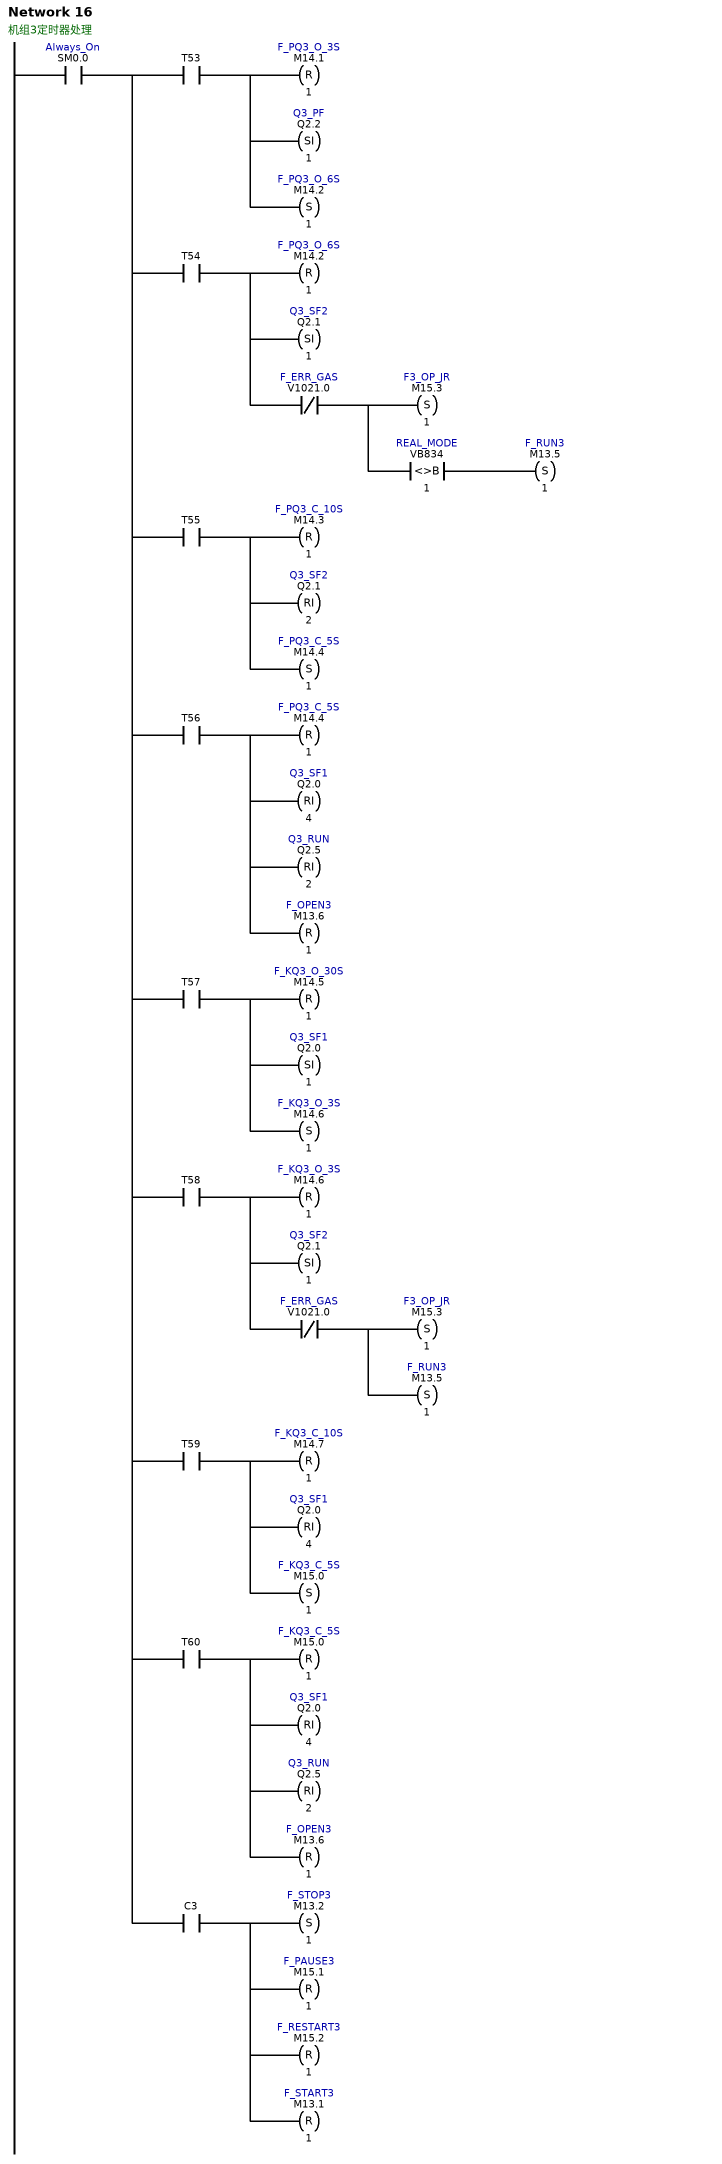
Network 16
// 机组3定时器处理
LD     Always_On:SM0.0
LPS
A      T53
R      F_PQ3_O_3S:M14.1, 1
SI     Q3_PF:Q2.2, 1
S      F_PQ3_O_6S:M14.2, 1
LRD
A      T54
R      F_PQ3_O_6S:M14.2, 1
SI     Q3_SF2:Q2.1, 1
AN     F_ERR_GAS:V1021.0
S      F3_OP_JR:M15.3, 1
AB<>   REAL_MODE:VB834, 1
S      F_RUN3:M13.5, 1
LRD
LPS
A      T55
R      F_PQ3_C_10S:M14.3, 1
RI     Q3_SF2:Q2.1, 2
S      F_PQ3_C_5S:M14.4, 1
LRD
A      T56
R      F_PQ3_C_5S:M14.4, 1
RI     Q3_SF1:Q2.0, 4
RI     Q3_RUN:Q2.5, 2
R      F_OPEN3:M13.6, 1
LPP
A      T57
R      F_KQ3_O_30S:M14.5, 1
SI     Q3_SF1:Q2.0, 1
S      F_KQ3_O_3S:M14.6, 1
LRD
A      T58
R      F_KQ3_O_3S:M14.6, 1
SI     Q3_SF2:Q2.1, 1
AN     F_ERR_GAS:V1021.0
S      F3_OP_JR:M15.3, 1
S      F_RUN3:M13.5, 1
LPP
LPS
A      T59
R      F_KQ3_C_10S:M14.7, 1
RI     Q3_SF1:Q2.0, 4
S      F_KQ3_C_5S:M15.0, 1
LRD
A      T60
R      F_KQ3_C_5S:M15.0, 1
RI     Q3_SF1:Q2.0, 4
RI     Q3_RUN:Q2.5, 2
R      F_OPEN3:M13.6, 1
LPP
A      C3
S      F_STOP3:M13.2, 1
R      F_PAUSE3:M15.1, 1
R      F_RESTART3:M15.2, 1
R      F_START3:M13.1, 1
